{attribute 'qualified_only'}
//{attribute 'strict'}
TYPE eSimState :
(
	no_sim := 0,
	Inserted := 1,
	active := 2,
	pin_fault := 3
);
END_TYPE

(* stored: Version 1.1.0.1, ProductVersion 3.1.4026.18
   DUT eSimState: Id {548202db-66b9-4551-a57d-35892e1ed5ed} *)
